(* CODESYS project FU_sConcat4.xml

Project tree, tasks and I/O mapping:
  function FU_sConcat4 [ST]
*)

// FU_sConcat4
//This functions combines four strings
// |**Version**|**Author**| **Date** |**Changes**
// | 1         | NSN      | 03-12-18 | Creation
FUNCTION FU_sConcat4 : STRING(255)
VAR_INPUT
	s1			:STRING(255);			//Input String1
	s2			:STRING(255);			//Input String2
	s3			:STRING(255);			//Input String3
	s4			:STRING(255);			//Input String4
END_VAR

FU_sConcat4BIBO(sOut:=ADR(FU_sConcat4),s1:=ADR(s1),s2:=ADR(s2),s3:=ADR(s3),s4:=ADR(s4),wOutSize:=255);

END_FUNCTION
